// TIA Portal V17 export
// export: Created 2023-03-06T02:05:27.7812381Z, ExportSetting WithDefaults, DisplayName Totally Integrated Automation Portal, DisplayVersion V17 Update 4, DisplayName TIA Portal Openness, DisplayVersion V17 Update 4, DisplayName TIA Portal Version Control Interface, DisplayVersion V17, DisplayName STEP 7 Professional, DisplayVersion V17 Update 4, DisplayName STEP 7 Safety, DisplayVersion V17, DisplayName WinCC Professional, DisplayVersion V17 Update 4
TYPE "MVSKID"
// stored: IsFailsafeCompliant false
   STRUCT
      iAssetSt : Int;
      iLine1DiscSt : Int;
      iLine1GroundSt : Int;
      iLine2DiscSt : Int;
      iLine2GroundSt : Int;
      iProt1DiscSt : Int;
      iProt1GroundSt : Int;
      iProt1CircBrkSt : Int;
      rTempTrafo : Real;
   END_STRUCT;
END_TYPE
